PROGRAM P4_05_Send
VAR
	fbAuditSend							:FB_PythonScript;
END_VAR
VAR // added by the converter: edge detectors and wires of the graphical bodies
    _rt1 : R_TRIG;
END_VAR

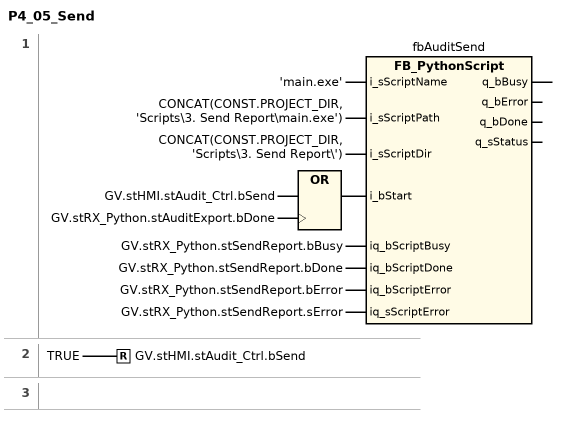
// NETWORK 1
_rt1(CLK := GV.stRX_Python.stAuditExport.bDone);
fbAuditSend(
    i_sScriptName := 'main.exe',
    i_sScriptPath := CONCAT(CONST.PROJECT_DIR,'Scripts\3. Send Report\main.exe'),
    i_sScriptDir := CONCAT(CONST.PROJECT_DIR,'Scripts\3. Send Report\'),
    i_bStart := GV.stHMI.stAudit_Ctrl.bSend OR _rt1.Q,
    iq_bScriptBusy := GV.stRX_Python.stSendReport.bBusy,
    iq_bScriptDone := GV.stRX_Python.stSendReport.bDone,
    iq_bScriptError := GV.stRX_Python.stSendReport.bError,
    iq_sScriptError := GV.stRX_Python.stSendReport.sError); // FB_PythonScript

// NETWORK 2
GV.stHMI.stAudit_Ctrl.bSend R= TRUE;

// NETWORK 3

END_PROGRAM

(* stored: Version 1.1.0.1
   POU P4_05_Send: Id {b653c921-2fb1-4678-804c-deeb49935df7}, SpecialFunc None *)
